{attribute 'qualified_only'}
{attribute 'strict'}
TYPE E_GEMMA :
(
    // Modos de la Guia de Estudio de los Modos de Marcha y Parada
    // Modes du Guide d'Etude des Modes de Marche et d'Arrêt
    // Modes of Study Guide of the Modes of Operating and Stopping

    // Procedimientos de parada [Les procédures d'arrets - Stop procedure
    A1, //  0: Parada en el estado inicial 
        //  0: Arrêt dans etat initial
        //  0: Stopped in the initial state
    A2, //  1: Parada solicitada a final de ciclo 
        //  1: Arret demandé en fin de cycle
        //  1: Requested end cycle stop
    A3, //  2: Parada solicitada en un estado determinado 
        //  2: Arret demande dans etat determine
        //  2: Requested particular state stop
    A4, //  3: Parada obtenida 
        //  3: Arret obtenu 
        //  3: Obteined stop
    A5, //  4: Preparacion para la recuperacion del fallo 
        //  4: Preparation pour remise en route apres defaillance
        //  4: Preparation for the recovery of the failure
    A6, //  5: Situando la PO en el estado inicial 
        //  5: Mise PO dans état initial 
        //  5: Set the PO in initial state
    A7, //  6: Situando la PO en un estado determinado 
        //  6: Mise PO dans état déterminé 
        //  6: Set the PO in a certain state

    // Procedimientos de funcionamiento 
    // Les procédures de fonctionnement 
    // Operating procedures
    F1, //  7: Produccion normal 
        //  7: Production normale 
        //  7: Normal operation
    F2, //  8: Secuencia de preparacion 
        //  8: Marche de preparation 
        //  8: Preparation sequence
    F3, //  9: Secuencia de finalizacion 
        //  9: Marche de cloture
        //  9: Ending sequence
    F4, // 10: Verificacion en desorden 
        // 10: Marche de verification dans le desordre 
        // 10: Verification with no order
    F5, // 11: Verificacion en orden 
        // 11: Marche de verification dans l'ordre 
        // 11: Verification whit order
    F6, // 12: Secuencia de prueba 
        // 12: Marche de test 
        // 12:Test sequence

    // Procedimientos de fallo 
    // es procédures en défaillances
    // Failure procedures
    D1, // 13: Parada de emergencia 
        // 13: Arret d'urgence 
        // 13: Emergency stop
    D2, // 14: Diagnostico y/o tratamiento de los fallos 
        // 14: Diagnostic et/ou traitement de la défaillance 
        // 14: Diagnosis and/or treatment of failures
    D3  // 15: Produccion a pesar de los fallos 
        // 15: Production tout de même 
        // 15: Production despite the failures
);
END_TYPE

(* stored: Version 1.1.0.1, ProductVersion 3.1.4024.9
   EnumerationTextList E_GEMMA: Id {00467c1d-a9d0-478a-9738-af8594f9212a} *)
